TEXTLIST MachineStateTextList
  1 = 'ManualState' | Chinese: '手动状态' | English: 'ManualState'
  2 = 'AutoState' | Chinese: '自动状态' | English: 'AutoState'
  3 = 'PauseState' | Chinese: '暂停状态' | English: 'PauseState'
  4 = 'StopState' | Chinese: '停止状态' | English: 'StopState'
  5 = 'ErrorState' | Chinese: '错误状态' | English: 'ErrorState'
  6 = 'HomeState' | Chinese: '回源状态' | English: 'HomeState'
   = ''
END_TEXTLIST

(* stored: Version 1.1.0.1, ProductVersion 3.1.4024.4
   TextList MachineStateTextList: Id {22405165-c187-4066-b85c-b31368cae7fa} *)
